TYPE TestTypeA :
STRUCT
	counter : INT := 0; (*second count until operator considered not alert*)
	(*TODO: alarm not implemented yet*)
	alarm : BOOL := FALSE; (*when counter reaches zero, this alarm is set to TRUE*)
END_STRUCT
END_TYPE

(* stored: Version 1.1.0.1, ProductVersion 3.1.4022.7
   DUT TestTypeA: Id {7b0e7fb8-7d0c-4904-9baf-2f3e0df9ef6e} *)
